// TIA Portal project "TrafficLight" (V18)

(* hardware
DEVICE "S7-1200 station_1"  S7-1200 Station
   slot 0: "Rack_0"  S7-1200 Rack  Rack  V1.0
   slot 1: "PLC_1"  CPU 1212C DC/DC/Rly  6ES7 212-1HE40-0XB0  V4.6
   slot 2: "DQ 8x24VDC _1"  SM 1222 DQ8 x 24VDC  6ES7 222-1BF32-0XB0  V2.0
DEVICE "TP1200 Comfort"  TP1200 Comfort
   slot 0: "TP1200 Comfort"  TP1200 Comfort  6AV2 124-0MC01-0AX0  16.0.0.0
   slot 1: "HMI_RT_3"  TP1200 Comfort  6AV2 124-0MC01-0AX0  16.0.0.0
   slot 5: "TP1200 Comfort._CP_1"  PROFINET Interface  16.0.0.0
      slot 1: "PROFINET Interface_1"  PROFINET Interface
         slot 1: "Port_1"  Port
         slot 2: "Port_2"  Port
   slot 7: "TP1200 Comfort.I/DP_CP_1"  MPI/DP Interface  16.0.0.0
*)

// ===== PLC "PLC_1"  CPU 1212C DC/DC/Rly =====

VAR_GLOBAL   // PLC tag table "Default tag table"
   "Clock_1Hz" AT %M0.5 : Bool;
END_VAR

VAR_GLOBAL   // PLC tag table "TrafficLightTags"
   "northLightGreen" AT %Q0.0 : Bool;
   "northLightYellow" AT %Q0.1 : Bool;
   "northLightRed" AT %Q0.2 : Bool;
   "southLightGreen" AT %Q0.3 : Bool;
   "southLightYellow" AT %Q0.4 : Bool;
   "southLightRed" AT %Q0.5 : Bool;
   "eastLightGreen" AT %Q1.0 : Bool;
   "eastLightYellow" AT %Q1.1 : Bool;
   "eastLightRed" AT %Q1.2 : Bool;
   "westLightGreen" AT %Q1.3 : Bool;
   "westLightYellow" AT %Q1.4 : Bool;
   "westLightRed" AT %Q1.5 : Bool;
   "systemFAULT" AT %M2.0 : Bool;
   "start_MEM_TAG" AT %M2.2 : Bool;
   "reset_MEM_TAG" AT %M2.1 : Bool;
   "start_Button_IN" AT %I0.0 : Bool;
   "reset_Button_IN" AT %I0.1 : Bool;
END_VAR

DATA_BLOCK "Intersection_DB"   // DB3
{ S7_Optimized_Access := 'TRUE' }
VERSION : 0.1
// stored: InstanceOfName Intersection
"Intersection"
BEGIN
END_DATA_BLOCK

FUNCTION_BLOCK "LightOperation"   // FB1, LAD
{ S7_Optimized_Access := 'TRUE' }
VERSION : 0.1
   VAR_INPUT
      start : Bool;
      reset : Bool;
   END_VAR
   VAR_OUTPUT
      lightGreen : Bool;
      lightYellow : Bool;
      lightRed : Bool;
      interlock : Bool;
   END_VAR
   VAR_IN_OUT
      fault : Bool;
   END_VAR
   VAR
      interlockRiseEdge : Bool;
      greenLightPulse : TP_TIME;
      yellowLightPulse : TP_TIME;
      greenLightFallEdge : Bool;
      yellowLightFallEdge : Bool;
      redlightRiseEdge : Bool;
   END_VAR
   VAR_TEMP   // added for the SCL form of the ladder/FBD networks
      _w1 : Bool;
      _w2 : Bool;
   END_VAR
BEGIN

REGION Network 1: Perform fault operation sequence when system is in fault and has not been reset
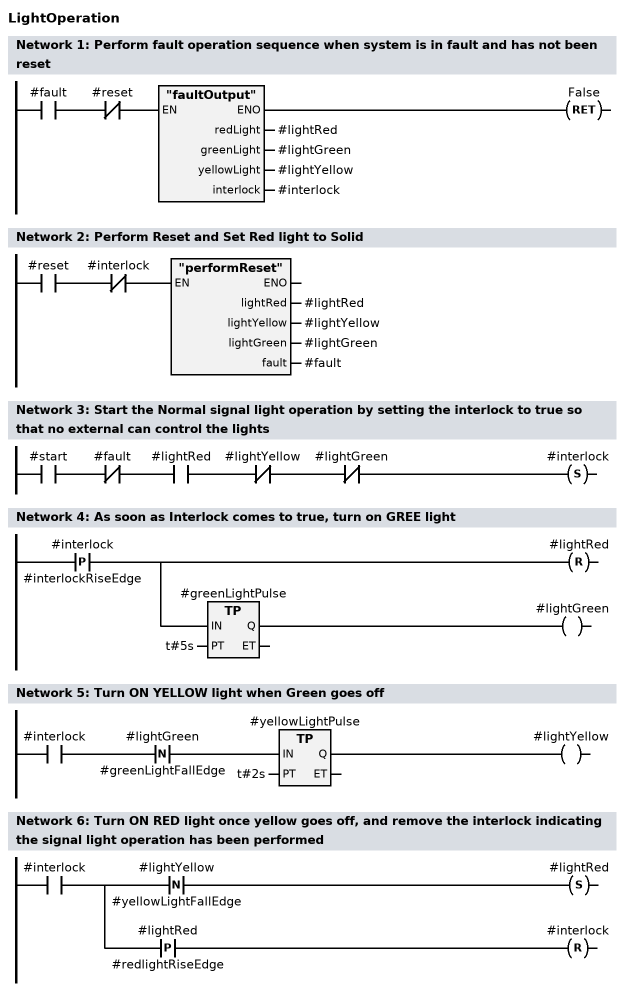
   "faultOutput"(EN := #fault AND NOT #reset,
                 redLight => #lightRed,
                 greenLight => #lightGreen,
                 yellowLight => #lightYellow,
                 interlock => #interlock,
                 ENO => #_w1);
   IF #_w1 THEN
       ENO := False;
       RETURN;
   END_IF;
END_REGION

REGION Network 2: Perform Reset and Set Red light to Solid
   RUNG wire#powerrail
      Contact( #reset )
      I_Contact( #interlock )
      "performReset"(lightRed => #lightRed, lightYellow => #lightYellow, lightGreen => #lightGreen, fault => #fault)
   END_RUNG
   // the same network as SCL:
   IF #reset AND NOT #interlock THEN
       "performReset"(lightRed => #lightRed,
                      lightYellow => #lightYellow,
                      lightGreen => #lightGreen,
                      fault => #fault);
   END_IF;
END_REGION

REGION Network 3: Start the Normal signal light operation by setting the interlock to true so that no external can control the lights
   RUNG wire#powerrail
      Contact( #start )
      I_Contact( #fault )
      Contact( #lightRed )
      I_Contact( #lightYellow )
      I_Contact( #lightGreen )
      S_Coil( #interlock )
   END_RUNG
   // the same network as SCL:
   IF #start AND NOT #fault AND #lightRed AND NOT #lightYellow AND NOT #lightGreen THEN
       #interlock := TRUE;
   END_IF;
END_REGION

REGION Network 4: As soon as Interlock comes to true, turn on GREE light
   #_w1 := #interlock AND NOT #interlockRiseEdge;   // rising edge of #interlock
   #interlockRiseEdge := #interlock;
   IF #_w1 THEN #lightRed := FALSE; END_IF;
   #greenLightPulse(IN := #_w1, PT := t#5s);   // TP
   #lightGreen := #greenLightPulse.Q;
END_REGION

REGION Network 5: Turn ON YELLOW light when Green goes off
   #_w1 := #interlock AND NOT #lightGreen AND #greenLightFallEdge;   // falling edge of #lightGreen
   #greenLightFallEdge := #lightGreen;
   #yellowLightPulse(IN := #_w1, PT := t#2s);   // TP
   #lightYellow := #yellowLightPulse.Q;
END_REGION

REGION Network 6: Turn ON RED light once yellow goes off, and remove the interlock indicating the signal light operation has been performed
   RUNG wire#powerrail
      Contact( #interlock )
      wire#w1
      N_Contact(operand := #lightYellow, bit := #yellowLightFallEdge)
      S_Coil( #lightRed )
   END_RUNG
   RUNG wire#w1
      P_Contact(operand := #lightRed, bit := #redlightRiseEdge)
      R_Coil( #interlock )
   END_RUNG
   // the same network as SCL:
   #_w1 := #interlock AND NOT #lightYellow AND #yellowLightFallEdge;   // falling edge of #lightYellow
   #yellowLightFallEdge := #lightYellow;
   IF #_w1 THEN #lightRed := TRUE; END_IF;
   #_w2 := #interlock AND #lightRed AND NOT #redlightRiseEdge;   // rising edge of #lightRed
   #redlightRiseEdge := #lightRed;
   IF #_w2 THEN #interlock := FALSE; END_IF;
END_REGION
END_FUNCTION_BLOCK

FUNCTION_BLOCK "Intersection"   // FB2, LAD
{ S7_Optimized_Access := 'TRUE' }
VERSION : 0.1
   VAR_OUTPUT
      northLightGreen : Bool;
      northLightYellow : Bool;
      northLightRed : Bool;
      southLightGreen : Bool;
      southLightYellow : Bool;
      southLightRed : Bool;
      eastLightGreen : Bool;
      eastLightYellow : Bool;
      eastLightRed : Bool;
      westLightGreen : Bool;
      westLightYellow : Bool;
      westLightRed : Bool;
   END_VAR
   VAR
      northLightOperation : "LightOperation";
      southLightOperation : "LightOperation";
      northInterlock : Bool;
      southInterlock : Bool;
      eastInterlock : Bool;
      westInterlock : Bool;
      eastLightOperation : "LightOperation";
      westLightOperation : "LightOperation";
      eastInterlockFallEdge : Bool;
      westInterlockFallEdge : Bool;
      northInterlockFallEdge : Bool;
      southInterlockFallEdge : Bool;
      northSouthONDelay : TON_TIME;
      eastWestONDelay : TON_TIME;
      startNorth : Bool;
      startSouth : Bool;
      startEast : Bool;
      startWest : Bool;
      startNSTimer : Bool;
      startEWTimer : Bool;
   END_VAR
   VAR_TEMP
      performRESET : Bool;
      performSTART : Bool;
   END_VAR
   VAR_TEMP   // added for the SCL form of the ladder/FBD networks
      _w1 : Bool;
      _w2 : Bool;
   END_VAR
BEGIN

REGION Network 1: Perform Reset or Start button event either through HMI button or PLC tag input
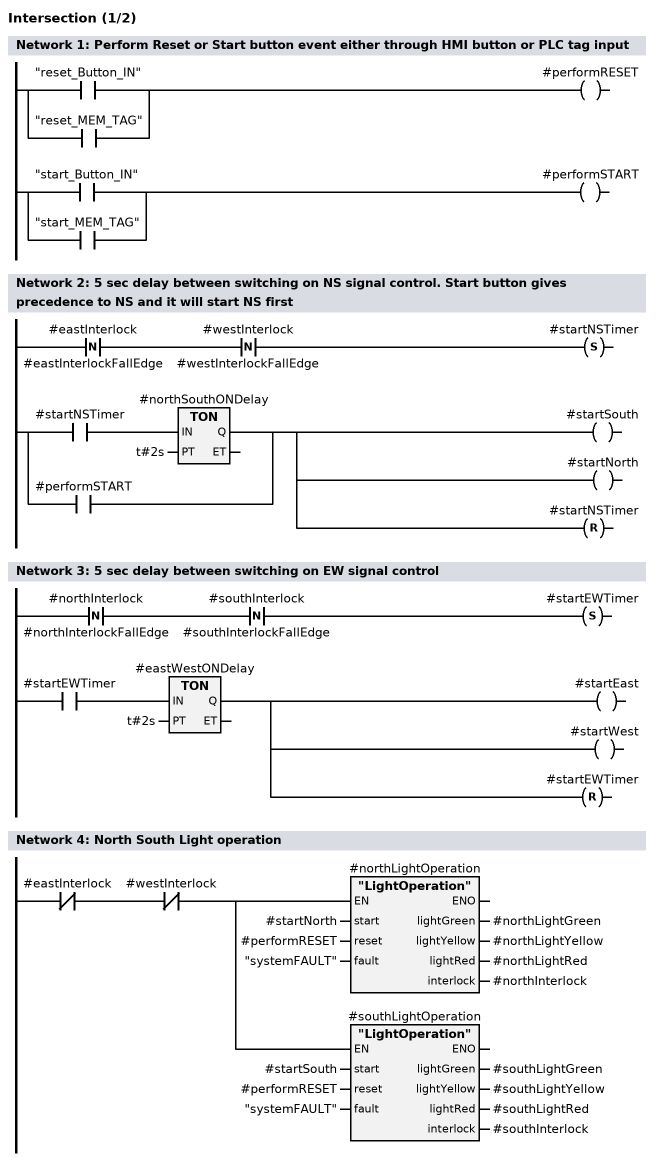
   RUNG wire#powerrail
      Contact( "reset_Button_IN" )
      wire#w1
      Coil( #performRESET )
   END_RUNG
   RUNG wire#powerrail
      Contact( "reset_MEM_TAG" )
   END_RUNG wire#w1
   RUNG wire#powerrail
      Contact( "start_Button_IN" )
      wire#w2
      Coil( #performSTART )
   END_RUNG
   RUNG wire#powerrail
      Contact( "start_MEM_TAG" )
   END_RUNG wire#w2
   // the same network as SCL:
   #performRESET := "reset_Button_IN" OR "reset_MEM_TAG";
   #performSTART := "start_Button_IN" OR "start_MEM_TAG";
END_REGION

REGION Network 2: 5 sec delay between switching on NS signal control. Start button gives precedence to NS and it will start NS first
   #_w1 := NOT #eastInterlock AND #eastInterlockFallEdge;   // falling edge of #eastInterlock
   #eastInterlockFallEdge := #eastInterlock;
   #_w2 := #_w1 AND NOT #westInterlock AND #westInterlockFallEdge;   // falling edge of #westInterlock
   #westInterlockFallEdge := #westInterlock;
   IF #_w2 THEN #startNSTimer := TRUE; END_IF;
   #northSouthONDelay(IN := #startNSTimer, PT := t#2s);   // TON
   #startSouth := #northSouthONDelay.Q OR #performSTART;
   #startNorth := #startSouth;
   IF #startSouth THEN #startNSTimer := FALSE; END_IF;
END_REGION

REGION Network 3: 5 sec delay between switching on EW signal control
   #_w1 := NOT #northInterlock AND #northInterlockFallEdge;   // falling edge of #northInterlock
   #northInterlockFallEdge := #northInterlock;
   #_w2 := #_w1 AND NOT #southInterlock AND #southInterlockFallEdge;   // falling edge of #southInterlock
   #southInterlockFallEdge := #southInterlock;
   IF #_w2 THEN #startEWTimer := TRUE; END_IF;
   #eastWestONDelay(IN := #startEWTimer, PT := t#2s);   // TON
   #startEast := #eastWestONDelay.Q;
   #startWest := #eastWestONDelay.Q;
   IF #eastWestONDelay.Q THEN #startEWTimer := FALSE; END_IF;
END_REGION

REGION Network 4: North South Light operation
   RUNG wire#powerrail
      I_Contact( #eastInterlock )
      I_Contact( #westInterlock )
      wire#w1
      #northLightOperation(start := #startNorth, reset := #performRESET, fault := "systemFAULT", lightGreen => #northLightGreen, lightYellow => #northLightYellow, lightRed => #northLightRed, interlock => #northInterlock)
   END_RUNG
   RUNG wire#w1
      #southLightOperation(start := #startSouth, reset := #performRESET, fault := "systemFAULT", lightGreen => #southLightGreen, lightYellow => #southLightYellow, lightRed => #southLightRed, interlock => #southInterlock)
   END_RUNG
   // the same network as SCL:
   IF NOT #eastInterlock AND NOT #westInterlock THEN
       #northLightOperation(start := #startNorth,   // "LightOperation"
                            reset := #performRESET,
                            fault := "systemFAULT",
                            lightGreen => #northLightGreen,
                            lightYellow => #northLightYellow,
                            lightRed => #northLightRed,
                            interlock => #northInterlock);
       #southLightOperation(start := #startSouth,   // "LightOperation"
                            reset := #performRESET,
                            fault := "systemFAULT",
                            lightGreen => #southLightGreen,
                            lightYellow => #southLightYellow,
                            lightRed => #southLightRed,
                            interlock => #southInterlock);
   END_IF;
END_REGION

REGION Network 5: East West Light operation
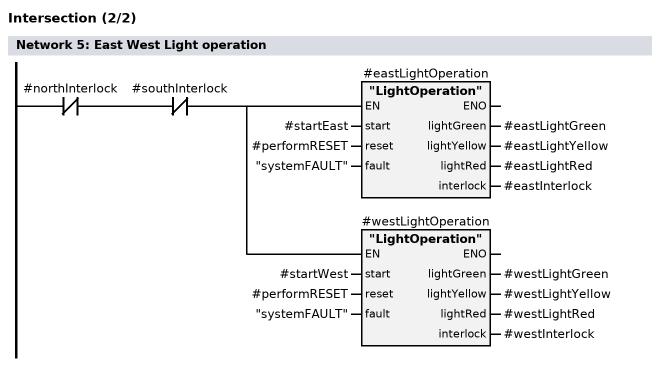
   RUNG wire#powerrail
      I_Contact( #northInterlock )
      I_Contact( #southInterlock )
      wire#w1
      #eastLightOperation(start := #startEast, reset := #performRESET, fault := "systemFAULT", lightGreen => #eastLightGreen, lightYellow => #eastLightYellow, lightRed => #eastLightRed, interlock => #eastInterlock)
   END_RUNG
   RUNG wire#w1
      #westLightOperation(start := #startWest, reset := #performRESET, fault := "systemFAULT", lightGreen => #westLightGreen, lightYellow => #westLightYellow, lightRed => #westLightRed, interlock => #westInterlock)
   END_RUNG
   // the same network as SCL:
   IF NOT #northInterlock AND NOT #southInterlock THEN
       #eastLightOperation(start := #startEast,   // "LightOperation"
                           reset := #performRESET,
                           fault := "systemFAULT",
                           lightGreen => #eastLightGreen,
                           lightYellow => #eastLightYellow,
                           lightRed => #eastLightRed,
                           interlock => #eastInterlock);
       #westLightOperation(start := #startWest,   // "LightOperation"
                           reset := #performRESET,
                           fault := "systemFAULT",
                           lightGreen => #westLightGreen,
                           lightYellow => #westLightYellow,
                           lightRed => #westLightRed,
                           interlock => #westInterlock);
   END_IF;
END_REGION
END_FUNCTION_BLOCK

FUNCTION "faultOutput" : Void   // FC1, LAD
{ S7_Optimized_Access := 'TRUE' }
VERSION : 0.1
   VAR_OUTPUT
      redLight : Bool;
      greenLight : Bool;
      yellowLight : Bool;
      interlock : Bool;
   END_VAR
BEGIN

REGION Network 1: Turn ON/OFF Red Light Every 1 second
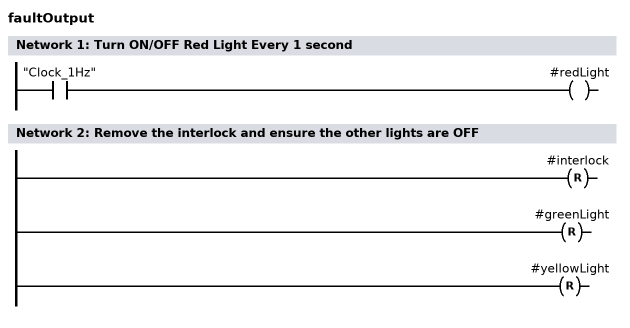
   RUNG wire#powerrail
      Contact( "Clock_1Hz" )
      Coil( #redLight )
   END_RUNG
   // the same network as SCL:
   #redLight := "Clock_1Hz";
END_REGION

REGION Network 2: Remove the interlock and ensure the other lights are OFF
   RUNG wire#powerrail
      R_Coil( #interlock )
   END_RUNG
   RUNG wire#powerrail
      R_Coil( #greenLight )
   END_RUNG
   RUNG wire#powerrail
      R_Coil( #yellowLight )
   END_RUNG
   // the same network as SCL:
   #interlock := FALSE;
   #greenLight := FALSE;
   #yellowLight := FALSE;
END_REGION
END_FUNCTION

FUNCTION "performReset" : Void   // FC2, LAD
TITLE = This block performs the RESET operation once the Reset button has been pressed
{ S7_Optimized_Access := 'TRUE' }
VERSION : 0.1
   VAR_OUTPUT
      lightRed : Bool;
      lightYellow : Bool;
      lightGreen : Bool;
      fault : Bool;
   END_VAR
BEGIN

REGION Network 1: Turn OFF Green
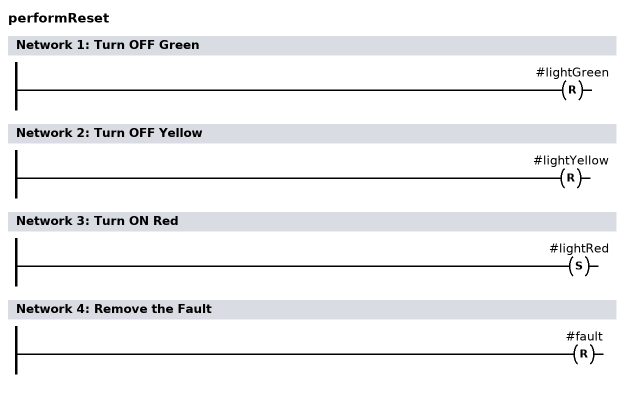
   RUNG wire#powerrail
      R_Coil( #lightGreen )
   END_RUNG
   // the same network as SCL:
   #lightGreen := FALSE;
END_REGION

REGION Network 2: Turn OFF Yellow
   RUNG wire#powerrail
      R_Coil( #lightYellow )
   END_RUNG
   // the same network as SCL:
   #lightYellow := FALSE;
END_REGION

REGION Network 3: Turn ON Red
   RUNG wire#powerrail
      S_Coil( #lightRed )
   END_RUNG
   // the same network as SCL:
   #lightRed := TRUE;
END_REGION

REGION Network 4: Remove the Fault
   RUNG wire#powerrail
      R_Coil( #fault )
   END_RUNG
   // the same network as SCL:
   #fault := FALSE;
END_REGION
END_FUNCTION

ORGANIZATION_BLOCK "Main"   // OB1, LAD, ProgramCycle
TITLE = "Main Program Sweep (Cycle)"
{ S7_Optimized_Access := 'TRUE' }
VERSION : 0.1
   VAR_INPUT
      Initial_Call : Bool;   // Initial call of this OB
      Remanence : Bool;   // =True, if remanent data are available
   END_VAR
BEGIN

REGION Network 1
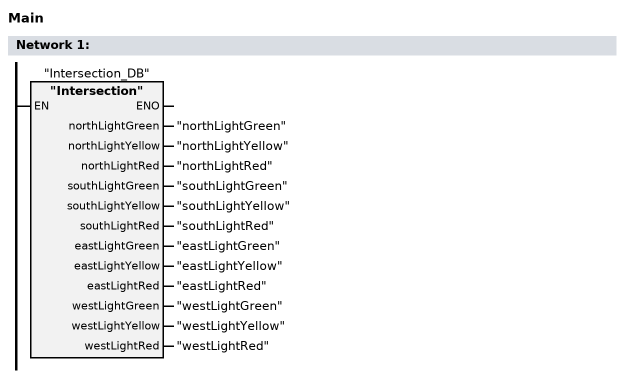
   RUNG wire#powerrail
      "Intersection_DB"(northLightGreen => "northLightGreen", northLightYellow => "northLightYellow", northLightRed => "northLightRed", southLightGreen => "southLightGreen", southLightYellow => "southLightYellow", southLightRed => "southLightRed", eastLightGreen => "eastLightGreen", eastLightYellow => "eastLightYellow", eastLightRed => "eastLightRed", westLightGreen => "westLightGreen", westLightYellow => "westLightYellow", westLightRed => "westLightRed")
   END_RUNG
   // the same network as SCL:
   "Intersection_DB"(northLightGreen => "northLightGreen",   // "Intersection"
                     northLightYellow => "northLightYellow",
                     northLightRed => "northLightRed",
                     southLightGreen => "southLightGreen",
                     southLightYellow => "southLightYellow",
                     southLightRed => "southLightRed",
                     eastLightGreen => "eastLightGreen",
                     eastLightYellow => "eastLightYellow",
                     eastLightRed => "eastLightRed",
                     westLightGreen => "westLightGreen",
                     westLightYellow => "westLightYellow",
                     westLightRed => "westLightRed");
END_REGION
END_ORGANIZATION_BLOCK

ORGANIZATION_BLOCK "Startup"   // OB100, LAD, Startup
TITLE = "Complete Restart"
{ S7_Optimized_Access := 'TRUE' }
VERSION : 0.1
   VAR_INPUT
      LostRetentive : Bool;   // True if retentive data are lost
      LostRTC : Bool;   // True if date and time are lost
   END_VAR
BEGIN

REGION Network 1
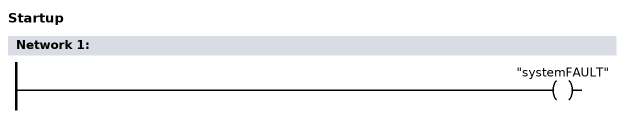
   RUNG wire#powerrail
      Coil( "systemFAULT" )
   END_RUNG
   // the same network as SCL:
   "systemFAULT" := TRUE;
END_REGION
END_ORGANIZATION_BLOCK

(* ===== HMI "HMI_RT_1" =====

ScreenModuleEditorView "North Signal Light Faceplate" 640x480
   GraphicView "Graphic view_3" at 10,10 size 70x142; Picture "PinClipart.com_attorney-clipart_1271995"
   Circle "Circle_4" at 26,18 size 39x39
      Appearance <- "redLight"
   Circle "Circle_5" at 26,62 size 39x39
      Appearance <- "yellowLight"
   Circle "Circle_6" at 26,106 size 39x39
      Appearance <- "greenLight"
*)

(* ===== HMI "HMI_RT_1" =====

ScreenModuleEditorView "South Signal Light Faceplate" 640x480
   GraphicView "Graphic view_1" at 10,10 size 70x142; Picture "south_facing_light"
   Circle "Circle_4" at 26,106 size 39x39
      Appearance <- "redLight"
   Circle "Circle_5" at 26,62 size 39x39
      Appearance <- "yellowLight"
   Circle "Circle_6" at 26,18 size 39x39
      Appearance <- "greenLight"
*)

(* ===== HMI "HMI_RT_1" =====

ScreenModuleEditorView "East Signal Light Faceplate" 640x480
   GraphicView "Graphic view_1" at 10,10 size 142x70; Picture "east_facing_light"
   Circle "Circle_4" at 106,26 size 39x39
      Appearance <- "redLight"
   Circle "Circle_5" at 62,26 size 39x39
      Appearance <- "yellowLight"
   Circle "Circle_6" at 18,26 size 39x39
      Appearance <- "greenLight"
*)

(* ===== HMI "HMI_RT_1" =====

ScreenModuleEditorView "West Signal Light Faceplate" 640x480
   GraphicView "Graphic view_1" at 10,10 size 142x70; Picture "west_facing_light"
   Circle "Circle_4" at 18,26 size 39x39
      Appearance <- "redLight"
   Circle "Circle_5" at 62,26 size 39x39
      Appearance <- "yellowLight"
   Circle "Circle_6" at 106,26 size 39x39
      Appearance <- "greenLight"
*)

(* ===== HMI "HMI_RT_3" =====
system functions are stored by id; their names below are inferred from use
connection "HMI_Connection_2": 
connection "HMI_Connection_1": ETHERNET, S7_1200_OMS

HMI tags "Template"
   "MainNavigationState" : Int, internal
   "SubNavigationState" : Int, internal
   "CurrentUserName" : WString[18], internal
   "DiagState" : Int, internal
   "PopUpBackground" : Bool, internal
   "UserName" : WString[20], internal
   "Password" : WString[20], internal
   "UserIsLoggedIn" : Bool, internal
   "CodeView" : Bool, internal
   "Brightness" : Int, internal
   "CurrentLanguage" : Bool, internal
   "CurrentRecipeName" : WString[30], internal
   "CurrentMachineState" : Int, internal
   "OptionPanelNavigationState" : Int, internal
   "ButtonDown" : Bool, internal
   "ThirdLevelNavigationState" : Int, internal
   "StartScreenName" : WString[60], internal
   "InScreenTabState" : Int, internal
   "DummyTagBool" : Bool, internal
   "DummyTagInt1" : Int, internal
   "DummyTagInt2" : Int, internal
   "DummyTagInt3" : Int, internal
   "DummyDeltaReal" : LReal, internal
   "DummTagReal1" : LReal, internal
   "DummyDeltaInt" : Int, internal

HMI tags "PLC_Tags"
   "eastLightGreen" : Bool = PLC eastLightGreen AT %Q1.0, 100 ms
   "eastLightRed" : Bool = PLC eastLightRed AT %Q1.2, 100 ms
   "eastLightYellow" : Bool = PLC eastLightYellow AT %Q1.1, 100 ms
   "northLightGreen" : Bool = PLC northLightGreen AT %Q0.0, 100 ms
   "northLightRed" : Bool = PLC northLightRed AT %Q0.2, 100 ms
   "northLightYellow" : Bool = PLC northLightYellow AT %Q0.1, 100 ms
   "reset_MEM_TAG" : Bool = PLC reset_MEM_TAG AT %M2.1, 100 ms
   "southLightGreen" : Bool = PLC southLightGreen AT %Q0.3, 100 ms
   "southLightRed" : Bool = PLC southLightRed AT %Q0.5, 100 ms
   "southLightYellow" : Bool = PLC southLightYellow AT %Q0.4, 100 ms
   "start_MEM_TAG" : Bool = PLC start_MEM_TAG AT %M2.2, 100 ms
   "systemFAULT" : Bool = PLC systemFAULT AT %M2.0, 100 ms
   "westLightGreen" : Bool = PLC westLightGreen AT %Q1.3, 100 ms
   "westLightRed" : Bool = PLC westLightRed AT %Q1.5, 100 ms
   "westLightYellow" : Bool = PLC westLightYellow AT %Q1.4, 100 ms

HMI tags "AnimationTags"
   "northGreenArrow" : Int, internal

text list "Machine State": 0 'Undefined / Kein Job'; 1 'Production / Produktion'; 2 'Startup / Anlauf'; 3 'Paused / Pausiert'; 4 'Stopped / Gestoppt'; 5 'Shutdown / Beenden'; 6 'Undefined / Unbekannt'

text list "timeRange": 1 'Hours / Stunden'; 2 'Days / Tage'; 3 'Weeks / Wochen'; 4 'Months / Monate'; 5 'Years / Jahre'

text list "MachineState_Farfield": 0..1 '???'; 1 'OK'; 2 'ERROR / FEHLER'; 3 'PAUSED / HALT'

text list "Foil Types": 0..1 '120 - 1mm - Transparent'; 1 '120 - 3mm - Transparent'; 2 '240 - 1mm - Transparent'; 3 '240 - 3mm - Transparent'

text list "FunctionState": 0 'Disabled / Deaktiviert'; 1 'Enabled / Aktiviert'

text list "GroundPos": 0 'No / Nein'; 1 'Yes / Ja'

text list "State": 0 'Off / Aus'; 1 'On / An'

graphic list "DiagState": 0 'DiagOkay'; 1 'DiagWarning_1'; 2 'DiagDefault'

graphic list "DiagState_1": 0 'DiagOkay_1'; 1 'DiagWarning'; 2 'DiagDefault'

graphic list "DiagState_2": 0 'DiagOkay_1'; 1 'DiagWarning'; 2 'DiagDefault'

graphic list "DiagState_3": 0 'DiagOkay_White'; 1 'DiagWarning_White'; 2 'Circle'

graphic list "State": 0..1 'OK'; 3 'Error'

graphic list "Machine": 1 'Grafik_Verpackung_Step1_Blink-off'; 2 'Grafik_Verpackung_Step2'; 3 'Grafik_Verpackung_Blink-on'; 6..7 'Grafik_Verpackung_Step1_Blink-off'

screen "10_Startscreen" 1280x800, template "01_One_Nav_Level"
   on GenerateScreen: "GetStartScreenName"(); "CheckCurrentUserName"(); SetTag("MainNavigationState", 1)
   GraphicView "Graphic view_2" at 0,0 size 1280x800; Picture "PopUpBackground"
      Visibility <- "PopUpBackground"
   GraphicView "Graphic view_1" at 0,104 size 1280x696; Picture "ChatGPT Image Oct 26, 2025, 03_33_37 PM(1)"
   ScreenModuleView "North Signal Light Faceplate_1" at 690,144 size 70x142; ScreenModuleType ""
      Guid_{11997190-6492} <- "northLightGreen"
      Guid_{11997190-6490} <- "northLightYellow"
      Guid_{11997190-6488} <- "northLightRed"
   ScreenModuleView "South Signal Light Faceplate_1" at 516,578 size 70x142; ScreenModuleType ""
      Guid_{11997190-6492} <- "southLightGreen"
      Guid_{11997190-6488} <- "southLightRed"
      Guid_{11997190-6490} <- "southLightYellow"
   ScreenModuleView "West Signal Light Faceplate_1" at 288,354 size 142x70; ScreenModuleType ""
      Guid_{11997190-6492} <- "westLightGreen"
      Guid_{11997190-6488} <- "westLightRed"
      Guid_{11997190-6490} <- "westLightYellow"
   ScreenModuleView "East Signal Light Faceplate_1" at 848,448 size 142x70; ScreenModuleType ""
      Guid_{11997190-6492} <- "eastLightGreen"
      Guid_{11997190-6488} <- "eastLightRed"
      Guid_{11997190-6490} <- "eastLightYellow"
   Button "Button_1" at 954,732 size 116x32; TextOff 'Start'
      on Press: function_b14e0dd5("start_MEM_TAG", 0)
      on Release: ResetBit("start_MEM_TAG")
   Button "Button_2" at 954,672 size 116x32; TextOff 'Reset'
      on Release: ResetBit("reset_MEM_TAG")
      on Press: function_b14e0dd5("reset_MEM_TAG", 0)
   Button "Button_3" at 953,614 size 116x32; TextOff 'Fault'
      on Click: SetBit("systemFAULT")
   Circle "Circle_1" at 1119,602 size 48x48
      Appearance <- "systemFAULT"
   GraphicView "Graphic view_3" at 681,354 size 94x219; Picture "up_arrow_3"
      Visibility <- "northLightGreen"
   GraphicView "Graphic view_4" at 511,331 size 94x219; Picture "down_arrow_1"
      Visibility <- "southLightGreen"
   GraphicView "Graphic view_5" at 418,453 size 395x94; Picture "right_arrow_1"
      Visibility <- "eastLightGreen"
   GraphicView "Graphic view_6" at 472,338 size 395x94; Picture "left_arrow_1"
      Visibility <- "westLightGreen"
   GraphicView "Graphic view_7" at 362,456 size 22x68; Picture "Stop_east"
      Visibility <- "eastLightGreen"
   GraphicView "Graphic view_8" at 690,602 size 68x22; Picture "Stop_north"
      Visibility <- "northLightGreen"
   GraphicView "Graphic view_9" at 888,354 size 22x68; Picture "Stop_west"
      Visibility <- "westLightGreen"
   GraphicView "Graphic view_10" at 516,238 size 68x22; Picture "Stop_south"
      Visibility <- "southLightGreen"
   GraphicView "Graphic view_11" at 988,132 size 173x165; Picture "unnamed_2"

screen "20_Messages" 1280x800, template "01_One_Nav_Level"
   on GenerateScreen: SetTag("MainNavigationState", 2)
   AlarmView "Alarm view_1" at 0,104 size 1280x695
   GraphicView "Graphic view_2" at 0,0 size 1280x800; Picture "PopUpBackground"
      Visibility <- "PopUpBackground"

screen "30_Diagnostics" 1280x800, template "01_One_Nav_Level"
   on GenerateScreen: SetTag("MainNavigationState", 3)
   SysDiagControl "System diagnostics view_1" at 0,104 size 1280x692
   GraphicView "Graphic view_2" at 0,0 size 1280x800; Picture "PopUpBackground"
      Visibility <- "PopUpBackground"
   GraphicView "gfxPrevScreenIcon" at 1240,763 size 24x24; Picture "PrevScreen_Icon"

screen "40_Settings" 1280x800, template "02_Settings"
   on GenerateScreen: SetTag("MainNavigationState", 4)
   Slider "Template_Slider_1" at 320,197 size 300x30; Caption 'SIMATIC'
      on Change: function_e4c2bb66("Brightness")
      ProcessValue <- "Brightness"
   TextField "Template_Text field_1" at 180,200 size 92x24; Text 'Brightness / Helligkeit'
   GraphicView "Graphic view_2" at 0,0 size 1280x800; Picture "PopUpBackground"
      Visibility <- "PopUpBackground"

Template "01_One_Nav_Level" 1280x800
   Gauge "gaugeDiagStateUpdate" at 566,2 size 50x50; CaptionText 'SIMATIC'
      on Change: "CheckDiagState"()
      ProcessValue <- "@DiagnosticsIndicatorTag"
   TextField "txtTitleBar" at 16,8 size 613x32; Text 'Traffic Light Control / Applikation'
   GraphicView "gfxNavigationIcon" at 1241,15 size 23x19; Picture "Hamburger_Icon"
   Button "btnNavigation" at 1224,0 size 56x48; TextOff 'Text'
      on Click: function_cf6f4242("GraphX_Slidein_Right", 1)
   Button "btnStartscreen" at 0,0 size 387x45; TextOff 'Text'
      on Click: "ActivateStartScreen"()
   TextField "txtStateHeadline" at 75,55 size 123x23; Text 'State / Status'
   TextField "txtRecipeHeadline" at 281,55 size 154x23; Text 'Current Recipe / Rezeptur'
   TextField "txtOperatorHeadline" at 527,55 size 129x23; Text 'Operator / Bediener'
   SymbolicIOField "ioState" at 75,72 size 119x30; TextOn '1'; TextOff '0'; TextList "Machine State"
      ProcessValue <- "CurrentMachineState"
   IOField "ioRecipe" at 281,72 size 158x30; FormatPattern ??????????????????????????????
      ProcessValue <- "CurrentRecipeName"
   IOField "ioOperator" at 527,72 size 126x30; FormatPattern ??????????????????
      ProcessValue <- "CurrentUserName"
   Button "btnState" at 202,56 size 40x40; TextOff '...'; PictureOff "More_Icon"
      on Click: "ShowOperatingModePopUp"()
   Button "btnRecipe" at 449,56 size 40x40; TextOff '...'; PictureOff "More_Icon"
      on Click: "ShowRecipePopUp"()
   Rectangle "rectState" at 0,48 size 56x56
      Appearance <- "CurrentMachineState"
   Rectangle "rectSystemDiagnosticsIndicator" at 1224,48 size 56x56
      Appearance <- "DiagState"
   GraphicIOField "gioDiagState" at 1236,60 size 32x32; PictureList "DiagState_3"
      ProcessValue <- "DiagState"
   Button "btnDiagState" at 1224,48 size 56x56; TextOff 'Text'
      on Click: ActivateScreen("30_Diagnostics", 0)
   Button "btnOperator" at 669,56 size 40x40; TextOff '...'; PictureOff "More_Icon"
      on Click: "ShowLoginPopUp"()
   TextField "txtOperatorHeadline_1" at 768,55 size 138x23; Text 'Date and Time / Datum und Uhrzeit'
   Button "btnOperator_1" at 995,56 size 40x40; TextOff '...'; PictureOff "More_Icon"; Authorization "User administration"
      on Click: function_f34a74f3()
   DateTimeField "Template_Date/time field_1" at 768,72 size 208x30

Template "02_Two_Nav_Levels" 1280x800
   GraphicView "gfxPrevScreenIcon" at 1240,763 size 24x24; Picture "PrevScreen_Icon"
   Button "btnSubNav1" at 0,752 size 144x48; TextOff 'Overview / Übersicht'
      on Click: SetTag("SubNavigationState", 1)
   Button "btnSubNav2" at 144,752 size 144x48; TextOff 'Module 1 / Modul 1'
      on Click: SetTag("SubNavigationState", 2)
   Button "btnSubNav3" at 288,752 size 144x48; TextOff 'Module 2 / Modul 2'
      on Click: SetTag("SubNavigationState", 3)
   Button "btnSubNav4" at 432,752 size 144x48; TextOff 'Module 3 / Modul 3'
      on Click: SetTag("SubNavigationState", 4)
   Button "btnSubNav5" at 576,752 size 144x48; TextOff 'Module 4 / Modul 4'
      on Click: SetTag("SubNavigationState", 5)
   Button "btnSubNav6" at 720,752 size 144x48; TextOff 'Module 5 / Modul 5'
      on Click: SetTag("SubNavigationState", 6)
   Button "btnSubNav7" at 864,752 size 144x48; TextOff 'Module 6 / Modul 6'
      on Click: SetTag("SubNavigationState", 7)
   Button "btnPreviousScreen" at 1224,751 size 56x48; TextOff 'Text'
      on Click: function_efd93a16()
   Gauge "gaugeDiagStateUpdate" at 566,2 size 50x50; CaptionText 'SIMATIC'
      on Change: "CheckDiagState"()
      ProcessValue <- "@DiagnosticsIndicatorTag"
   TextField "txtTitleBar" at 16,8 size 495x32; Text 'Traffic Light Control / Applikation'
   GraphicView "gfxNavigationIcon" at 1241,15 size 23x19; Picture "Hamburger_Icon"
   Button "btnNavigation" at 1224,0 size 56x48; TextOff 'Text'
      on Click: function_cf6f4242("GraphX_Slidein_Right", 1)
   TextField "txtStateHeadline" at 75,55 size 123x23; Text 'State / Status'
   TextField "txtRecipeHeadline" at 281,55 size 154x23; Text 'Current Recipe / Rezeptur'
   TextField "txtOperatorHeadline" at 527,55 size 129x23; Text 'Operator / Bediener'
   SymbolicIOField "ioState" at 75,72 size 119x30; TextOn '1'; TextOff '0'; TextList "Machine State"
      ProcessValue <- "CurrentMachineState"
   IOField "ioRecipe" at 281,72 size 158x30; FormatPattern ??????????????????????????????
      ProcessValue <- "CurrentRecipeName"
   IOField "ioOperator" at 527,72 size 126x30; FormatPattern ??????????????????
      ProcessValue <- "CurrentUserName"
   Button "btnState" at 202,56 size 40x40; TextOff '...'; PictureOff "More_Icon"
      on Click: "ShowOperatingModePopUp"()
   Button "btnRecipe" at 449,56 size 40x40; TextOff '...'; PictureOff "More_Icon"
      on Click: "ShowRecipePopUp"()
   Rectangle "rectState" at 0,48 size 56x56
      Appearance <- "CurrentMachineState"
   Rectangle "rectSystemDiagnosticsIndicator" at 1224,48 size 56x56
      Appearance <- "DiagState"
   GraphicIOField "gioDiagState" at 1236,60 size 32x32; PictureList "DiagState_3"
      ProcessValue <- "DiagState"
   Button "btnDiagState" at 1224,48 size 56x56; TextOff 'Text'
      on Click: ActivateScreen("30_Diagnostics", 0)
   Button "btnOperator" at 669,56 size 40x40; TextOff '...'; PictureOff "More_Icon"
      on Click: "ShowLoginPopUp"()
   TextField "txtOperatorHeadline_1" at 768,55 size 138x23; Text 'Date and Time / Datum und Uhrzeit'
   DateTimeField "Template_Date/time field_1" at 768,72 size 208x30
   Button "btnOperator_1" at 995,56 size 40x40; TextOff '...'; Authorization "User administration"; PictureOff "More_Icon"
      on Click: function_f34a74f3()
   Button "btnStartscreen" at 0,0 size 250x45; TextOff 'Text'
      on Click: "ActivateStartScreen"()
   Button "btnSubNavActive1" at 0,752 size 144x48; TextOff 'Overview / Übersicht'
      Visibility <- "SubNavigationState"
   Button "btnSubNavActive2" at 144,752 size 144x48; TextOff 'Module 1 / Modul 1'
      Visibility <- "SubNavigationState"
   Button "btnSubNavActive3" at 288,752 size 144x48; TextOff 'Module 2 / Modul 2'
      Visibility <- "SubNavigationState"
   Button "btnSubNavActive4" at 432,752 size 144x48; TextOff 'Module 3 / Modul 3'
      Visibility <- "SubNavigationState"
   Button "btnSubNavActive5" at 576,752 size 144x48; TextOff 'Module 4 / Modul 4'
      Visibility <- "SubNavigationState"
   Button "btnSubNavActive6" at 720,752 size 144x48; TextOff 'Module 5 / Modul 5'
      Visibility <- "SubNavigationState"
   Button "btnSubNavActive7" at 864,752 size 144x48; TextOff 'Module 6 / Modul 6'
      Visibility <- "SubNavigationState"
   Rectangle "rectIndicatorActive1" at 0,795 size 144x5
      Visibility <- "SubNavigationState"
   Rectangle "rectIndicatorActive2" at 144,795 size 144x5
      Visibility <- "SubNavigationState"
   Rectangle "rectIndicatorActive3" at 288,795 size 144x5
      Visibility <- "SubNavigationState"
   Rectangle "rectIndicatorActive4" at 432,795 size 144x5
      Visibility <- "SubNavigationState"
   Rectangle "rectIndicatorActive5" at 576,795 size 144x5
      Visibility <- "SubNavigationState"
   Rectangle "rectIndicatorActive6" at 720,795 size 144x5
      Visibility <- "SubNavigationState"
   Rectangle "rectIndicatorActive7" at 864,795 size 144x5
      Visibility <- "SubNavigationState"

Template "02_Two_Nav_Levels_Large_Text" 1280x800
   TextField "txtNextBackup1" at 16,120 size 232x24; Text 'Option 1'
   IOField "ioTargetPath1" at 16,152 size 236x24; FormatPattern ??????????????????????????????????????????????????
   TextField "txtNextBackup2" at 16,228 size 232x24; Text 'Option 2'
   IOField "ioTargetPath2" at 16,260 size 236x24; FormatPattern ??????????????????????????????????????????????????
   TextField "txtNextBackup3" at 16,336 size 232x24; Text 'Option 3'
   IOField "ioTargetPath3" at 16,368 size 236x24; FormatPattern ??????????????????????????????????????????????????
   TextField "txtNextBackup4" at 16,443 size 232x24; Text 'Option 4'
   IOField "ioTargetPath4" at 16,475 size 236x24; FormatPattern ??????????????????????????????????????????????????
   TextField "txtNextBackup5" at 16,551 size 232x24; Text 'Option 5'
   IOField "ioTargetPath5" at 16,583 size 236x24; FormatPattern ??????????????????????????????????????????????????
   TextField "txtNextBackup6" at 16,659 size 232x24; Text 'Option 6'
   IOField "ioTargetPath6" at 16,691 size 236x24; FormatPattern ??????????????????????????????????????????????????
   Button "btnSubNavigation1" at 0,104 size 264x109; TextOff 'Text'
      on Click: SetTag("ThirdLevelNavigationState", 1)
   Button "btnSubNavigation2" at 0,212 size 264x109; TextOff 'Text'
      on Click: SetTag("ThirdLevelNavigationState", 2)
   Button "btnSubNavigation3" at 0,320 size 264x109; TextOff 'Text'
      on Click: SetTag("ThirdLevelNavigationState", 3)
   Button "btnSubNavigation4" at 0,428 size 264x109; TextOff 'Text'
      on Click: SetTag("ThirdLevelNavigationState", 4)
   Button "btnSubNavigation5" at 0,536 size 264x109; TextOff 'Text'
      on Click: SetTag("ThirdLevelNavigationState", 5)
   Button "btnSubNavigation6" at 0,644 size 264x109; TextOff 'Text'
      on Click: SetTag("ThirdLevelNavigationState", 6)
   Gauge "gaugeDiagStateUpdate" at 566,2 size 50x50; CaptionText 'SIMATIC'
      on Change: "CheckDiagState"()
      ProcessValue <- "@DiagnosticsIndicatorTag"
   TextField "txtTitleBar" at 16,8 size 495x32; Text 'Traffic Light Control / Applikation'
   GraphicView "gfxNavigationIcon" at 1241,15 size 23x19; Picture "Hamburger_Icon"
   Button "btnNavigation" at 1224,0 size 56x48; TextOff 'Text'
      on Click: function_cf6f4242("GraphX_Slidein_Right", 1)
   Button "btnStartscreen" at 0,0 size 250x45; TextOff 'Text'
      on Click: "ActivateStartScreen"()
   TextField "txtStateHeadline" at 75,55 size 123x23; Text 'State / Status'
   TextField "txtRecipeHeadline" at 281,55 size 154x23; Text 'Current Recipe / Rezeptur'
   TextField "txtOperatorHeadline" at 527,55 size 129x23; Text 'Operator / Bediener'
   SymbolicIOField "ioState" at 75,72 size 119x30; TextOn '1'; TextOff '0'; TextList "Machine State"
      ProcessValue <- "CurrentMachineState"
   IOField "ioRecipe" at 281,72 size 158x30; FormatPattern ??????????????????????????????
      ProcessValue <- "CurrentRecipeName"
   IOField "ioOperator" at 527,72 size 126x30; FormatPattern ??????????????????
      ProcessValue <- "CurrentUserName"
   Button "btnState" at 202,56 size 40x40; TextOff '...'; PictureOff "More_Icon"
      on Click: "ShowOperatingModePopUp"()
   Button "btnRecipe" at 449,56 size 40x40; TextOff '...'; PictureOff "More_Icon"
      on Click: "ShowRecipePopUp"()
   Rectangle "rectState" at 0,48 size 56x56
      Appearance <- "CurrentMachineState"
   Rectangle "rectSystemDiagnosticsIndicator" at 1224,48 size 56x56
      Appearance <- "DiagState"
   GraphicIOField "gioDiagState" at 1236,60 size 32x32; PictureList "DiagState_3"
      ProcessValue <- "DiagState"
   Button "btnDiagState" at 1224,48 size 56x56; TextOff 'Text'
      on Click: ActivateScreen("30_Diagnostics", 0)
   Button "btnOperator" at 669,56 size 40x40; TextOff '...'; PictureOff "More_Icon"
      on Click: "ShowLoginPopUp"()
   TextField "txtOperatorHeadline_1" at 768,55 size 138x23; Text 'Date and Time / Datum und Uhrzeit'
   DateTimeField "Template_Date/time field_1" at 768,72 size 208x30
   Button "btnOperator_1" at 995,56 size 40x40; TextOff '...'; Authorization "User administration"; PictureOff "More_Icon"
      on Click: function_f34a74f3()
   Rectangle "rectSubNavigation1" at 0,104 size 264x109
      Appearance <- "ThirdLevelNavigationState"
   Rectangle "rectSubNavigation2" at 0,212 size 264x109
      Appearance <- "ThirdLevelNavigationState"
   Rectangle "rectSubNavigation3" at 0,320 size 264x109
      Appearance <- "ThirdLevelNavigationState"
   Rectangle "rectSubNavigation4" at 0,428 size 264x109
      Appearance <- "ThirdLevelNavigationState"
   GraphicView "gfxPrevScreenIcon" at 1240,763 size 24x24; Picture "PrevScreen_Icon"
   TextField "txtCurrentStateInfo" at 16,764 size 505x24; Text 'Optional Text about current state / Optionaler text mit aktuellem Status'
   Rectangle "rectSubNavigation4_1" at 0,536 size 264x109
      Appearance <- "ThirdLevelNavigationState"
   Rectangle "rectSubNavigation4_2" at 0,644 size 264x108
      Appearance <- "ThirdLevelNavigationState"
   Button "btnPreviousScreen" at 1224,752 size 56x48; TextOff 'Text'
      on Click: function_efd93a16()

Template "02_Two_Nav_Levels_Text" 1280x800
   Button "btnSubNav1" at 0,146 size 144x56; TextOn 'Item 1'; TextOff 'Item 1'
      on Click: SetTag("SubNavigationState", 1)
   Button "btnSubNav2" at 0,201 size 144x56; TextOn 'Item 2'; TextOff 'Item 2'
      on Click: SetTag("SubNavigationState", 2)
   Button "btnSubNav3" at 0,256 size 144x60; TextOn 'Item 3'; TextOff 'Item 3'
      on Click: SetTag("SubNavigationState", 3)
   Button "btnSubNav4" at 0,315 size 144x60; TextOn 'Item 4'; TextOff 'Item 4'
      on Click: SetTag("SubNavigationState", 4)
   Button "btnSubNav5" at 0,374 size 144x60; TextOn 'Item 5'; TextOff 'Item 5'
      on Click: SetTag("SubNavigationState", 4)
   GraphicView "gfxRuntimeStop" at 61,763 size 23x28; Picture "Power_dark"
   Button "btnRuntimeStop" at 0,752 size 144x48; TextOff 'Text'
      on Click: StopRuntime(0)
   Button "btnSubNavActive1" at 0,146 size 144x56; TextOff 'Item 1'
      Visibility <- "SubNavigationState"
   Button "btnSubNavActive2" at 0,201 size 144x56; TextOff 'Item 2'
      Visibility <- "SubNavigationState"
   Button "btnSubNavActive3" at 0,256 size 144x60; TextOff 'Item 3'
      Visibility <- "SubNavigationState"
   Button "btnSubNavActive4" at 0,315 size 144x60; TextOff 'Item 4'
      Visibility <- "SubNavigationState"
   Button "btnSubNavActive5" at 0,374 size 144x60; TextOn 'Item 5'; TextOff 'Item 5'
      Visibility <- "SubNavigationState"
   Rectangle "rectIndicatorActive1" at 0,146 size 5x56
      Visibility <- "SubNavigationState"
   Rectangle "rectIndicatorActive2" at 0,201 size 5x56
      Visibility <- "SubNavigationState"
   Rectangle "rectIndicatorActive3" at 0,256 size 5x60
      Visibility <- "SubNavigationState"
   Rectangle "rectIndicatorActive4" at 0,315 size 5x60
      Visibility <- "SubNavigationState"
   Rectangle "rectIndicatorActive5" at 0,374 size 5x60
      Visibility <- "SubNavigationState"
   Gauge "gaugeDiagStateUpdate" at 566,2 size 50x50; CaptionText 'SIMATIC'
      on Change: "CheckDiagState"()
      ProcessValue <- "@DiagnosticsIndicatorTag"
   TextField "txtTitleBar" at 16,8 size 495x32; Text 'Traffic Light Control / Applikation'
   GraphicView "gfxNavigationIcon" at 1241,15 size 23x19; Picture "Hamburger_Icon"
   Button "btnNavigation" at 1224,0 size 56x48; TextOff 'Text'
      on Click: function_cf6f4242("GraphX_Slidein_Right", 1)
   Button "btnStartscreen" at 0,0 size 250x45; TextOff 'Text'
      on Click: "ActivateStartScreen"()
   TextField "txtStateHeadline" at 75,55 size 123x23; Text 'State / Status'
   TextField "txtRecipeHeadline" at 281,55 size 154x23; Text 'Current Recipe / Rezeptur'
   TextField "txtOperatorHeadline" at 527,55 size 129x23; Text 'Operator / Bediener'
   SymbolicIOField "ioState" at 75,72 size 119x30; TextOn '1'; TextOff '0'; TextList "Machine State"
      ProcessValue <- "CurrentMachineState"
   IOField "ioRecipe" at 281,72 size 158x30; FormatPattern ??????????????????????????????
      ProcessValue <- "CurrentRecipeName"
   IOField "ioOperator" at 527,72 size 126x30; FormatPattern ??????????????????
      ProcessValue <- "CurrentUserName"
   Button "btnState" at 202,56 size 40x40; TextOff '...'; PictureOff "More_Icon"
      on Click: "ShowOperatingModePopUp"()
   Button "btnRecipe" at 449,56 size 40x40; TextOff '...'; PictureOff "More_Icon"
      on Click: "ShowRecipePopUp"()
   Rectangle "rectState" at 0,48 size 56x56
      Appearance <- "CurrentMachineState"
   Rectangle "rectSystemDiagnosticsIndicator" at 1224,48 size 56x56
      Appearance <- "DiagState"
   GraphicIOField "gioDiagState" at 1236,60 size 32x32; PictureList "DiagState_3"
      ProcessValue <- "DiagState"
   Button "btnDiagState" at 1224,48 size 56x56; TextOff 'Text'
      on Click: ActivateScreen("30_Diagnostics", 0)
   Button "btnOperator" at 669,56 size 40x40; TextOff '...'; PictureOff "More_Icon"
      on Click: "ShowLoginPopUp"()
   TextField "txtOperatorHeadline_1" at 768,55 size 138x23; Text 'Date and Time / Datum und Uhrzeit'
   DateTimeField "Template_Date/time field_1" at 768,72 size 208x30
   Button "btnOperator_1" at 995,56 size 40x40; TextOff '...'; Authorization "User administration"; PictureOff "More_Icon"
      on Click: function_f34a74f3()

Template "03_Three_Nav_Levels" 1280x800
   Gauge "gaugeDiagStateUpdate" at 566,2 size 50x50; CaptionText 'SIMATIC'
      on Change: "CheckDiagState"()
      ProcessValue <- "@DiagnosticsIndicatorTag"
   TextField "txtTitleBar" at 16,8 size 495x32; Text 'Traffic Light Control / Applikation'
   GraphicView "gfxNavigationIcon" at 1241,15 size 23x19; Picture "Hamburger_Icon"
   Button "btnNavigation" at 1224,0 size 56x48; TextOff 'Text'
      on Click: function_cf6f4242("GraphX_Slidein_Right", 1)
   TextField "txtStateHeadline" at 75,55 size 123x23; Text 'State / Status'
   TextField "txtRecipeHeadline" at 281,55 size 154x23; Text 'Current Recipe / Rezeptur'
   TextField "txtOperatorHeadline" at 527,55 size 129x23; Text 'Operator / Bediener'
   SymbolicIOField "ioState" at 75,72 size 119x30; TextOn '1'; TextOff '0'; TextList "Machine State"
      ProcessValue <- "CurrentMachineState"
   IOField "ioRecipe" at 281,72 size 158x30; FormatPattern ??????????????????????????????
      ProcessValue <- "CurrentRecipeName"
   IOField "ioOperator" at 527,72 size 126x30; FormatPattern ??????????????????
      ProcessValue <- "CurrentUserName"
   Button "btnState" at 202,56 size 40x40; TextOff '...'; PictureOff "More_Icon"
      on Click: "ShowOperatingModePopUp"()
   Button "btnRecipe" at 449,56 size 40x40; TextOff '...'; PictureOff "More_Icon"
      on Click: "ShowRecipePopUp"()
   Rectangle "rectState" at 0,48 size 56x56
      Appearance <- "CurrentMachineState"
   Rectangle "rectSystemDiagnosticsIndicator" at 1224,48 size 56x56
      Appearance <- "DiagState"
   GraphicIOField "gioDiagState" at 1236,60 size 32x32; PictureList "DiagState_3"
      ProcessValue <- "DiagState"
   Button "btnDiagState" at 1224,48 size 56x56; TextOff 'Text'
      on Click: ActivateScreen("30_Diagnostics", 0)
   Button "btnOperator" at 669,56 size 40x40; TextOff '...'; PictureOff "More_Icon"
      on Click: "ShowLoginPopUp"()
   TextField "txtOperatorHeadline_1" at 768,55 size 138x23; Text 'Date and Time / Datum und Uhrzeit'
   DateTimeField "Template_Date/time field_1" at 768,72 size 208x30
   Button "btnOperator_1" at 995,56 size 40x40; TextOff '...'; Authorization "User administration"; PictureOff "More_Icon"
      on Click: function_f34a74f3()
   Button "btnStartscreen" at 0,0 size 250x45; TextOff 'Text'
      on Click: "ActivateStartScreen"()
   Button "btnThirdLevel4btnOff1" at 0,104 size 56x163; TextOff 'Text'
   Button "btnThirdLevel4btnOff2" at 0,266 size 56x162; TextOff 'Text'
   Button "btnThirdLevel4btnOff3" at 0,427 size 56x163; TextOff 'Text'
   Button "btnThirdLevel4btnOff4" at 0,589 size 56x163; TextOff 'Text'
   Button "btnThirdLevel4btnOn1" at 0,266 size 56x161; TextOff 'Text'
      Visibility <- "ThirdLevelNavigationState"
   Button "btnThirdLevel4btnOn2" at 0,104 size 56x161; TextOff 'Text'
      Visibility <- "ThirdLevelNavigationState"
   Button "btnThirdLevel4btnOn3" at 0,428 size 56x161; TextOff 'Text'
      Visibility <- "ThirdLevelNavigationState"
   Button "btnThirdLevel4btnOn4" at 0,590 size 56x162; TextOff 'Text'
      Visibility <- "ThirdLevelNavigationState"
   Rectangle "rectIndicator4btnActive1" at 0,104 size 5x161
      Visibility <- "ThirdLevelNavigationState"
   Rectangle "rectIndicator4btnActive2" at 0,266 size 5x161
      Visibility <- "ThirdLevelNavigationState"
   Rectangle "rectIndicator4btnActive3" at 0,428 size 5x161
      Visibility <- "ThirdLevelNavigationState"
   Rectangle "rectIndicator4btnActive4" at 0,590 size 5x162
      Visibility <- "ThirdLevelNavigationState"
   Button "btnSubNavActive1" at 0,752 size 144x48; TextOff 'Overview / Übersicht'
      Visibility <- "SubNavigationState"
   Button "btnSubNavActive2" at 144,752 size 144x48; TextOff 'Module 1 / Modul 1'
      Visibility <- "SubNavigationState"
   Button "btnSubNavActive3" at 288,752 size 144x48; TextOff 'Module 2 / Modul 2'
      Visibility <- "SubNavigationState"
   Button "btnSubNavActive4" at 432,752 size 144x48; TextOff 'Module 3 / Modul 3'
      Visibility <- "SubNavigationState"
   Button "btnSubNavActive5" at 576,752 size 144x48; TextOff 'Module 4 / Modul 4'
      Visibility <- "SubNavigationState"
   Button "btnSubNavActive6" at 720,752 size 144x48; TextOff 'Module 5 / Modul 5'
      Visibility <- "SubNavigationState"
   Button "btnSubNavActive7" at 864,752 size 144x48; TextOff 'Module 6 / Modul 6'
      Visibility <- "SubNavigationState"
   Rectangle "rectIndicatorActive1" at 0,795 size 144x5
      Visibility <- "SubNavigationState"
   Rectangle "rectIndicatorActive2" at 144,795 size 144x5
      Visibility <- "SubNavigationState"
   Rectangle "rectIndicatorActive3" at 288,795 size 144x5
      Visibility <- "SubNavigationState"
   Rectangle "rectIndicatorActive4" at 432,795 size 144x5
      Visibility <- "SubNavigationState"
   Rectangle "rectIndicatorActive5" at 576,795 size 144x5
      Visibility <- "SubNavigationState"
   Rectangle "rectIndicatorActive6" at 720,795 size 144x5
      Visibility <- "SubNavigationState"
   Rectangle "rectIndicatorActive7" at 864,795 size 144x5
      Visibility <- "SubNavigationState"
   GraphicView "gfxPrevScreenIcon" at 1240,763 size 24x24; Picture "PrevScreen_Icon"
   Button "btnSubNav1" at 0,752 size 144x48; TextOff 'Overview / Übersicht'
      on Click: SetTag("SubNavigationState", 1)
   Button "btnSubNav2" at 144,752 size 144x48; TextOff 'Module 1 / Modul 1'
      on Click: SetTag("SubNavigationState", 2)
   Button "btnSubNav3" at 288,752 size 144x48; TextOff 'Module 2 / Modul 2'
      on Click: SetTag("SubNavigationState", 3)
   Button "btnSubNav4" at 432,752 size 144x48; TextOff 'Module 3 / Modul 3'
      on Click: SetTag("SubNavigationState", 4)
   Button "btnSubNav5" at 576,752 size 144x48; TextOff 'Module 4 / Modul 4'
      on Click: SetTag("SubNavigationState", 5)
   Button "btnSubNav6" at 720,752 size 144x48; TextOff 'Module 5 / Modul 5'
      on Click: SetTag("SubNavigationState", 6)
   Button "btnSubNav7" at 864,752 size 144x48; TextOff 'Module 6 / Modul 6'
      on Click: SetTag("SubNavigationState", 7)
   Button "btnPreviousScreen" at 1224,751 size 56x48; TextOff 'Text'
      on Click: function_efd93a16()

Template "03_Three_Nav_Levels_w_OptionPanel" 1280x800
   Gauge "gaugeDiagStateUpdate" at 566,2 size 50x50; CaptionText 'SIMATIC'
      on Change: "CheckDiagState"()
      ProcessValue <- "@DiagnosticsIndicatorTag"
   TextField "txtTitleBar" at 16,8 size 495x32; Text 'Traffic Light Control / Applikation'
   GraphicView "gfxNavigationIcon" at 1241,15 size 23x19; Picture "Hamburger_Icon"
   Button "btnNavigation" at 1224,0 size 56x48; TextOff 'Text'
      on Click: function_cf6f4242("GraphX_Slidein_Right", 1)
   TextField "txtStateHeadline" at 75,55 size 123x23; Text 'State / Status'
   TextField "txtRecipeHeadline" at 281,55 size 154x23; Text 'Current Recipe / Rezeptur'
   TextField "txtOperatorHeadline" at 527,55 size 129x23; Text 'Operator / Bediener'
   SymbolicIOField "ioState" at 75,72 size 119x30; TextOn '1'; TextOff '0'; TextList "Machine State"
      ProcessValue <- "CurrentMachineState"
   IOField "ioRecipe" at 281,72 size 158x30; FormatPattern ??????????????????????????????
      ProcessValue <- "CurrentRecipeName"
   IOField "ioOperator" at 527,72 size 126x30; FormatPattern ??????????????????
      ProcessValue <- "CurrentUserName"
   Button "btnState" at 202,56 size 40x40; TextOff '...'; PictureOff "More_Icon"
      on Click: "ShowOperatingModePopUp"()
   Button "btnRecipe" at 449,56 size 40x40; TextOff '...'; PictureOff "More_Icon"
      on Click: "ShowRecipePopUp"()
   Rectangle "rectState" at 0,48 size 56x56
      Appearance <- "CurrentMachineState"
   Rectangle "rectSystemDiagnosticsIndicator" at 1224,48 size 56x56
      Appearance <- "DiagState"
   GraphicIOField "gioDiagState" at 1236,60 size 32x32; PictureList "DiagState_3"
      ProcessValue <- "DiagState"
   Button "btnDiagState" at 1224,48 size 56x56; TextOff 'Text'
      on Click: ActivateScreen("30_Diagnostics", 0)
   Button "btnOperator" at 669,56 size 40x40; TextOff '...'; PictureOff "More_Icon"
      on Click: "ShowLoginPopUp"()
   TextField "txtOperatorHeadline_1" at 768,55 size 138x23; Text 'Date and Time / Datum und Uhrzeit'
   DateTimeField "Template_Date/time field_1" at 768,72 size 208x30
   Button "btnOperator_1" at 995,56 size 40x40; TextOff '...'; Authorization "User administration"; PictureOff "More_Icon"
      on Click: function_f34a74f3()
   Button "btnStartscreen" at 0,0 size 250x45; TextOff 'Text'
      on Click: "ActivateStartScreen"()
   Button "btnThirdLevel4btnOff1" at 0,104 size 56x163; TextOff 'Text'
   Button "btnThirdLevel4btnOff2" at 0,266 size 56x162; TextOff 'Text'
   Button "btnThirdLevel4btnOff3" at 0,427 size 56x163; TextOff 'Text'
   Button "btnThirdLevel4btnOff4" at 0,589 size 56x163; TextOff 'Text'
   Button "btnThirdLevel4btnOn1" at 0,266 size 56x161; TextOff 'Text'
      Visibility <- "ThirdLevelNavigationState"
   Button "btnThirdLevel4btnOn2" at 0,104 size 56x161; TextOff 'Text'
      Visibility <- "ThirdLevelNavigationState"
   Button "btnThirdLevel4btnOn3" at 0,428 size 56x161; TextOff 'Text'
      Visibility <- "ThirdLevelNavigationState"
   Button "btnThirdLevel4btnOn4" at 0,590 size 56x162; TextOff 'Text'
      Visibility <- "ThirdLevelNavigationState"
   Rectangle "rectIndicator4btnActive1" at 0,104 size 5x161
      Visibility <- "ThirdLevelNavigationState"
   Rectangle "rectIndicator4btnActive2" at 0,266 size 5x161
      Visibility <- "ThirdLevelNavigationState"
   Rectangle "rectIndicator4btnActive3" at 0,428 size 5x161
      Visibility <- "ThirdLevelNavigationState"
   Rectangle "rectIndicator4btnActive4" at 0,590 size 5x162
      Visibility <- "ThirdLevelNavigationState"
   Button "btnOptionbtn1" at 1224,104 size 56x648; TextOff 'Text'; PictureOn "ManFunctions_Off"; PictureOff "ManFunctions_Off"
      on Click: "ShowOptionPanelPopUp"()
   GraphicView "gfxPrevScreenIcon" at 1240,763 size 24x24; Picture "PrevScreen_Icon"
   Button "btnSubNav1" at 0,752 size 144x48; TextOff 'Overview / Übersicht'
      on Click: SetTag("SubNavigationState", 1)
   Button "btnSubNav2" at 144,752 size 144x48; TextOff 'Module 1 / Modul 1'
      on Click: SetTag("SubNavigationState", 2)
   Button "btnSubNav3" at 288,752 size 144x48; TextOff 'Module 2 / Modul 2'
      on Click: SetTag("SubNavigationState", 3)
   Button "btnSubNav4" at 432,752 size 144x48; TextOff 'Module 3 / Modul 3'
      on Click: SetTag("SubNavigationState", 4)
   Button "btnSubNav5" at 576,752 size 144x48; TextOff 'Module 4 / Modul 4'
      on Click: SetTag("SubNavigationState", 5)
   Button "btnSubNav6" at 720,752 size 144x48; TextOff 'Module 5 / Modul 5'
      on Click: SetTag("SubNavigationState", 6)
   Button "btnSubNav7" at 864,752 size 144x48; TextOff 'Module 6 / Modul 6'
      on Click: SetTag("SubNavigationState", 7)
   Button "btnPreviousScreen" at 1224,751 size 56x48; TextOff 'Text'
      on Click: function_efd93a16()
   Button "btnSubNavActive1" at 0,752 size 144x48; TextOff 'Overview / Übersicht'
      Visibility <- "SubNavigationState"
   Button "btnSubNavActive2" at 144,752 size 144x48; TextOff 'Module 1 / Modul 1'
      Visibility <- "SubNavigationState"
   Button "btnSubNavActive3" at 288,752 size 144x48; TextOff 'Module 2 / Modul 2'
      Visibility <- "SubNavigationState"
   Button "btnSubNavActive4" at 432,752 size 144x48; TextOff 'Module 3 / Modul 3'
      Visibility <- "SubNavigationState"
   Button "btnSubNavActive5" at 576,752 size 144x48; TextOff 'Module 4 / Modul 4'
      Visibility <- "SubNavigationState"
   Button "btnSubNavActive6" at 720,752 size 144x48; TextOff 'Module 5 / Modul 5'
      Visibility <- "SubNavigationState"
   Button "btnSubNavActive7" at 864,752 size 144x48; TextOff 'Module 6 / Modul 6'
      Visibility <- "SubNavigationState"
   Rectangle "rectIndicatorActive1" at 0,795 size 144x5
      Visibility <- "SubNavigationState"
   Rectangle "rectIndicatorActive2" at 144,795 size 144x5
      Visibility <- "SubNavigationState"
   Rectangle "rectIndicatorActive3" at 288,795 size 144x5
      Visibility <- "SubNavigationState"
   Rectangle "rectIndicatorActive4" at 432,795 size 144x5
      Visibility <- "SubNavigationState"
   Rectangle "rectIndicatorActive5" at 576,795 size 144x5
      Visibility <- "SubNavigationState"
   Rectangle "rectIndicatorActive6" at 720,795 size 144x5
      Visibility <- "SubNavigationState"
   Rectangle "rectIndicatorActive7" at 864,795 size 144x5
      Visibility <- "SubNavigationState"

Template "02_Settings" 1280x800
   Button "btnSubNav1" at 0,184 size 136x56; TextOn 'Display'; TextOff 'Display'
      on Click: SetTag("SubNavigationState", 1)
   GraphicView "gfxRuntimeStop" at 57,763 size 23x28; Picture "Power_dark"
   Button "btnRuntimeStop" at 0,752 size 136x48; TextOff 'Text'
      on Click: StopRuntime(0)
   Button "btnSubNavActive1" at 0,184 size 136x56; TextOn 'Display'; TextOff 'Display'
      Visibility <- "SubNavigationState"
   Rectangle "rectIndicatorActive1" at 0,184 size 5x56
      Visibility <- "SubNavigationState"
   Gauge "gaugeDiagStateUpdate" at 566,2 size 50x50; CaptionText 'SIMATIC'
      on Change: "CheckDiagState"()
      ProcessValue <- "@DiagnosticsIndicatorTag"
   TextField "txtTitleBar" at 16,8 size 613x32; Text 'Traffic Light Control / Applikation'
   GraphicView "gfxNavigationIcon" at 1241,15 size 23x19; Picture "Hamburger_Icon"
   Button "btnNavigation" at 1224,0 size 56x48; TextOff 'Text'
      on Click: function_cf6f4242("GraphX_Slidein_Right", 1)
   Button "btnStartscreen" at 0,0 size 387x45; TextOff 'Text'
      on Click: "ActivateStartScreen"()
   TextField "txtStateHeadline" at 75,55 size 123x23; Text 'State / Status'
   TextField "txtRecipeHeadline" at 281,55 size 154x23; Text 'Current Recipe / Rezeptur'
   TextField "txtOperatorHeadline" at 527,55 size 129x23; Text 'Operator / Bediener'
   SymbolicIOField "ioState" at 75,72 size 119x30; TextOn '1'; TextOff '0'; TextList "Machine State"
      ProcessValue <- "CurrentMachineState"
   IOField "ioRecipe" at 281,72 size 158x30; FormatPattern ??????????????????????????????
      ProcessValue <- "CurrentRecipeName"
   IOField "ioOperator" at 527,72 size 126x30; FormatPattern ??????????????????
      ProcessValue <- "CurrentUserName"
   Button "btnState" at 202,56 size 40x40; TextOff '...'; PictureOff "More_Icon"
      on Click: "ShowOperatingModePopUp"()
   Button "btnRecipe" at 449,56 size 40x40; TextOff '...'; PictureOff "More_Icon"
      on Click: "ShowRecipePopUp"()
   Rectangle "rectState" at 0,48 size 56x56
      Appearance <- "CurrentMachineState"
   Rectangle "rectSystemDiagnosticsIndicator" at 1224,48 size 56x56
      Appearance <- "DiagState"
   GraphicIOField "gioDiagState" at 1236,60 size 32x32; PictureList "DiagState_3"
      ProcessValue <- "DiagState"
   Button "btnDiagState" at 1224,48 size 56x56; TextOff 'Text'
      on Click: ActivateScreen("30_Diagnostics", 0)
   Button "btnOperator" at 669,56 size 40x40; TextOff '...'; PictureOff "More_Icon"
      on Click: "ShowLoginPopUp"()
   TextField "txtOperatorHeadline_1" at 768,55 size 138x23; Text 'Date and Time / Datum und Uhrzeit'
   DateTimeField "Template_Date/time field_1" at 768,72 size 208x30
   Button "btnOperator_1" at 995,56 size 40x40; TextOff '...'; Authorization "User administration"; PictureOff "More_Icon"
      on Click: function_f34a74f3()

PopupScreen "Template_Logon" 320x352
   on ClearScreen: ResetBit("PopUpBackground")
   on GenerateScreen: SetBit("PopUpBackground")
   TextField "Template_Text field_1" at 16,0 size 215x40; Text 'Login'
   Button "Button_2" at 16,240 size 288x40; TextOn 'LOGIN / ANMELDEN'; TextOff 'LOGIN / ANMELDEN'
      on Click: function_a9b89908("Password", "UserName"); function_efd93a16("Template_Logon", 0, 0, 0, -1, 1)
   IOField "I/O field_1" at 16,84 size 288x40; FormatPattern ??????????????????????????????
      ProcessValue <- "UserName"
   TextField "Text field_1" at 16,56 size 288x24; Text 'User Name / Name'
   IOField "I/O field_2" at 16,168 size 288x40; FormatPattern ??????????????????????????????
      ProcessValue <- "Password"
   TextField "Text field_2" at 16,140 size 288x24; Text 'Password / Passwort'
   Button "Button_1" at 16,296 size 288x40; TextOn 'CLOSE / SCHLIESSEN'; TextOff 'CLOSE / SCHLIESSEN'
      on Click: function_efd93a16("Template_Logon", 0, 0, 0, -1, 1)
      on Press: function_b14e0dd5("ButtonDown", 0)
      Appearance <- "ButtonDown"

PopupScreen "Template_Logon_Logoff" 320x352
   on ClearScreen: ResetBit("PopUpBackground")
   on GenerateScreen: SetBit("PopUpBackground")
   TextField "Template_Text field_1" at 16,0 size 215x40; Text 'Login'
   Button "Button_2" at 16,240 size 136x40; TextOn 'LOG OFF / ABMELDEN'; TextOff 'LOG OFF / ABMELDEN'
      on Click: function_f23ef4c9()
   IOField "I/O field_1" at 16,84 size 288x40; FormatPattern ??????????????????????????????
      ProcessValue <- "UserName"
   TextField "Text field_1" at 16,56 size 288x24; Text 'User Name / Name'
   IOField "I/O field_2" at 16,168 size 288x40; FormatPattern ??????????????????????????????
      ProcessValue <- "Password"
   TextField "Text field_2" at 16,140 size 288x24; Text 'Password / Passwort'
   Button "Button_1" at 16,296 size 288x40; TextOn 'CLOSE / SCHLIESSEN'; TextOff 'CLOSE / SCHLIESSEN'
      on Click: function_efd93a16("Template_Logon_Logoff", 0, 0, 0, -1, 1)
      on Press: function_b14e0dd5("ButtonDown", 0)
      Appearance <- "ButtonDown"
   Button "Button_3" at 168,240 size 136x40; TextOn 'LOGIN / ANMELDEN'; TextOff 'LOGIN / ANMELDEN'
      on Click: function_a9b89908("Password", "UserName"); function_efd93a16("Template_Logon_Logoff", 0, 0, 0, -1, 1)

PopupScreen "Template_Operating_Mode" 424x360
   on ClearScreen: ResetBit("PopUpBackground")
   on GenerateScreen: SetBit("PopUpBackground")
   TextField "Template_Text field_1" at 14,0 size 336x40; Text 'Operating Mode / Betriebsmodus'
   Button "Button_1" at 80,304 size 260x40; TextOn 'CLOSE / SCHLIESSEN'; TextOff 'CLOSE / SCHLIESSEN'
      on Click: function_efd93a16("Template_Operating_Mode", 0, 0, 0, -1, 1)
      on Press: function_b14e0dd5("ButtonDown", 0)
      Appearance <- "ButtonDown"
   Button "Button_2" at 352,66 size 40x40; TextOff 'Text'; PictureOff "More_Icon"; PictureOn "More_Icon"
   Button "Button_3" at 352,130 size 40x40; TextOff 'Text'; PictureOff "More_Icon"; PictureOn "More_Icon"
   Button "Button_4" at 28,210 size 82x48; TextOff 'Start'
      on Press: function_b14e0dd5("start_MEM_TAG", 0)
      on Release: ResetBit("start_MEM_TAG")
   Button "Button_5" at 123,210 size 82x48; TextOff 'Stop'
      on Click: SetBit("systemFAULT")
      on Release: ResetBit("systemFAULT")
   Button "Button_6" at 218,210 size 82x48; TextOff 'Reset'
      on Press: function_b14e0dd5("reset_MEM_TAG", 0)
      on Release: ResetBit("reset_MEM_TAG")
   Button "Button_7" at 314,210 size 82x48; TextOff 'Hold'
   TextField "txtParameter7_3" at 32,63 size 163x24; Text 'Current Mode'
   IOField "ioParameter17_3" at 32,81 size 301x40; FormatPattern ?????????????????????????
   TextField "txtParameter7_1" at 32,127 size 163x24; Text 'Current State'
   IOField "ioParameter17_1" at 32,145 size 301x40; FormatPattern ?????????????????????????

PopupScreen "Template_Recipe" 700x420
   on ClearScreen: ResetBit("PopUpBackground")
   on GenerateScreen: SetBit("PopUpBackground")
   TextField "Template_Text field_1" at 14,0 size 500x40; Text 'Recipe / Rezeptur'
   Button "Button_1" at 220,364 size 260x40; TextOn 'CLOSE / SCHLIESSEN'; TextOff 'CLOSE / SCHLIESSEN'
      on Click: function_efd93a16("Template_Recipe", 0, 0, 0, -1, 1)
      on Press: function_b14e0dd5("ButtonDown", 0)
      Appearance <- "ButtonDown"
   RecipeView "Rezepturanzeige_1" at 0,40 size 700x320

PopupScreen "OptionPanel_4_Buttons" 390x648
   Button "btnCloseOptionPanel" at 0,0 size 40x648; TextOff 'CLOSE'; PictureOff "Jog_Forward"
      on Press: function_efd93a16("OptionPanel_4_Buttons", 0, 0, 0, 2, 2)
   TextField "txtOptionPanel" at 108,16 size 260x40; Text 'Option Panel Title / Titel Option Panel'
   Button "btnOption1" at 80,72 size 240x40; TextOff 'Option 1 / Move to Home Position'
   Button "btnOption2" at 80,128 size 240x40; TextOff 'Option 2 / Move to Home Position'
   Button "btnOption3" at 80,184 size 240x40; TextOff 'Option 3 / RESET'
   Button "btnOption4" at 80,240 size 240x40; TextOff 'Option 4 / RESET'
   GraphicView "gvOptionPanel" at 80,30 size 18x12; Picture "ManFunctions_Off"

SlideinScreen "GraphX_Slidein_Right" 220x800
   Button "Button_1" at 0,78 size 220x60; TextOn 'Menu Item 1'; TextOff 'Startscreen / Startseite'
      on Click: ActivateScreen("10_Startscreen", 0)
      Appearance <- "MainNavigationState"
   Button "Button_2" at 0,140 size 220x60; TextOn 'Menu Item 2'; TextOff 'Messages / Meldungen'
      on Click: ActivateScreen("20_Messages", 0)
      Appearance <- "MainNavigationState"
   Button "Button_3" at 0,201 size 220x60; TextOn 'Menu Item 3'; TextOff 'Diagnostics / Diagnose'
      on Click: ActivateScreen("30_Diagnostics", 0)
      Appearance <- "MainNavigationState"
   Rectangle "Rectangle_1" at 214,78 size 6x60
      Visibility <- "MainNavigationState"
   Rectangle "Rectangle_2" at 214,140 size 6x60
      Visibility <- "MainNavigationState"
   Rectangle "Rectangle_3" at 214,201 size 6x60
      Visibility <- "MainNavigationState"
   Button "Button_4" at 0,262 size 220x60; TextOn 'Menu Item 4'; TextOff 'Settings / Einstellungen'
      on Click: ActivateScreen("40_Settings", 0)
      Appearance <- "MainNavigationState"
   Rectangle "Rectangle_4" at 214,262 size 6x60
      Visibility <- "MainNavigationState"

VB script "ActivateAlarmControlScreen"
   bec8f1e5-2ab1-45f6-ad91-1d37c469eb91 20_Messages,0

VB script "ActivateStartScreen"
   HmiRuntime.BaseScreenName = SmartTags("StartScreenName")

VB script "CheckCurrentLanguage"
   If HmiRuntime.Language = 1031 Then 'German
   	SmartTags("CurrentLanguage") = 0
   	ElseIf HmiRuntime.Language = 1033 Then 'English US
   	SmartTags("CurrentLanguage") = 1
   End If
   
   	

VB script "CheckCurrentUserName"
   If SmartTags("CurrentUserName") = "" Or SmartTags("CurrentUserName") = "User Name" Or SmartTags("CurrentUserName") = "Benutzer" Then
     
     If HmiRuntime.Language = 1031 Then 'Germany
       SmartTags("CurrentUserName") = "Benutzer"
       
     ElseIf HmiRuntime.Language = 1033 Then 'English US
       SmartTags("CurrentUserName") = "User Name"
     End If
     
     SmartTags("UserIsLoggedIn") = False
   Else
     If SmartTags("CurrentUserName") <> "User Name" And SmartTags("CurrentUserName") <> "Benutzer" Then
       SmartTags("UserIsLoggedIn") = True  
     End If
   End If

VB script "CheckDiagState"
   If SmartTags("@DiagnosticsIndicatorTag") = 1 Then
   	SmartTags("DiagState") = 1
   Else
   	SmartTags("DiagState") = 0
   End If

VB script "GetStartScreenName"
   SmartTags("StartScreenName") = HmiRuntime.BaseScreenName

VB script "ShowLoginPopUp"
   efd93a16-2665-4b85-bcb9-25eddcb7b6f4 Template_Logon_Logoff,480,110,$3$hmiOn$,$3$hmiAnimationOff$,$3$hmiFast$

VB script "ShowOperatingModePopUp"
   efd93a16-2665-4b85-bcb9-25eddcb7b6f4 Template_Operating_Mode,428,110,$3$hmiOn$,$3$hmiAnimationOff$,$3$hmiFast$

VB script "ShowOptionPanelPopUp"
   efd93a16-2665-4b85-bcb9-25eddcb7b6f4 OptionPanel_4_Buttons, 890, 110, $3$hmiOn$, $3$hmiRight$, $3$hmiFast$

VB script "ShowRecipePopUp"
   efd93a16-2665-4b85-bcb9-25eddcb7b6f4 Template_Recipe,290,110,$3$hmiOn$,$3$hmiAnimationOff$,$3$hmiFast$

scheduled task "User Name"
   on Action: function_f41c6f6c("CurrentUserName"); "CheckCurrentUserName"()
*)